(* Logix 5000 project; controller Turck_IOLink_All_Full_AOIs_V0_1 vendor 1 type 14 code 176 rev 32.11; software revision 32.00; part 7 of 7 *)
(* tags used below, declared in another part *)
   Port : INT;
   Write_Application_Specific_Tag : BOOL;
   Universal_IOLink_Info : Universal_IOLink_Info;
   StartupDone : BOOL;
   Done : DINT;
   Error : DINT;
   Active : DINT;
   Pending : DINT;
   Pending_or_Active : DINT;
   MyTicketNum : DINT[32];
   DoneCount : DINT;
   Status : DINT;
   ErrorCount : DINT;
   Prev_Vendor_ID : INT;
   Write_ONS : DINT;
   WriteRequest : DINT;
(* Universal_Device_Info, continued *)

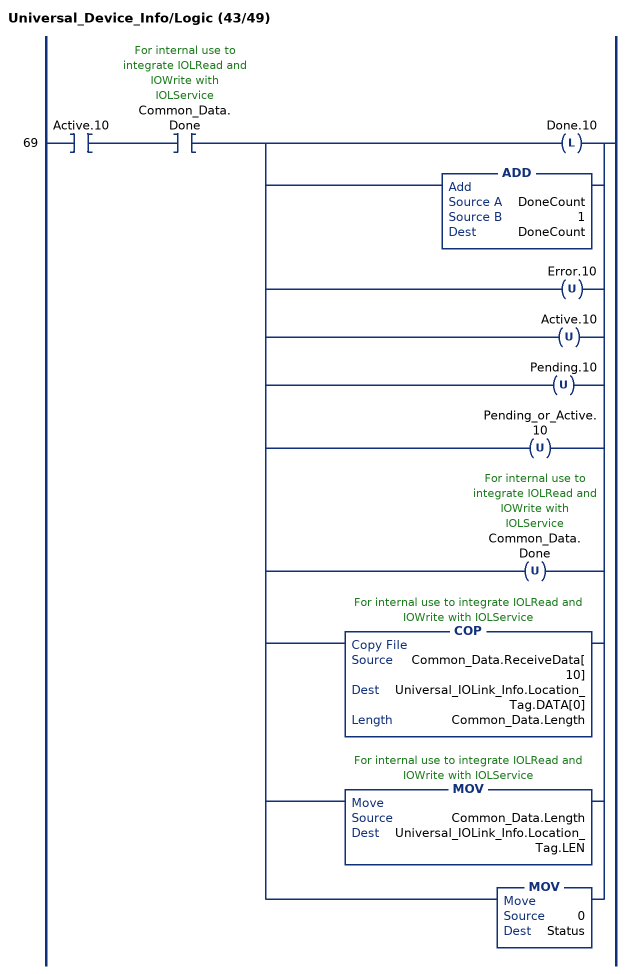
   [picture p146: Universal_Device_Info/Logic rungs 69-69]
   69: XIC(Active.10)XIC(Common_Data.Done)[OTL(Done.10) ,ADD(DoneCount,1,DoneCount) ,OTU(Error.10) ,OTU(Active.10) ,OTU(Pending.10) ,OTU(Pending_or_Active.10) ,OTU(Common_Data.Done) ,COP(Common_Data.ReceiveData[10],Universal_IOLink_Info.Location_Tag.DATA[0],Common_Data.Length) ,MOV(Common_Data.Length,Universal_IOLink_Info.Location_Tag.LEN) ,MOV(0,Status) ];
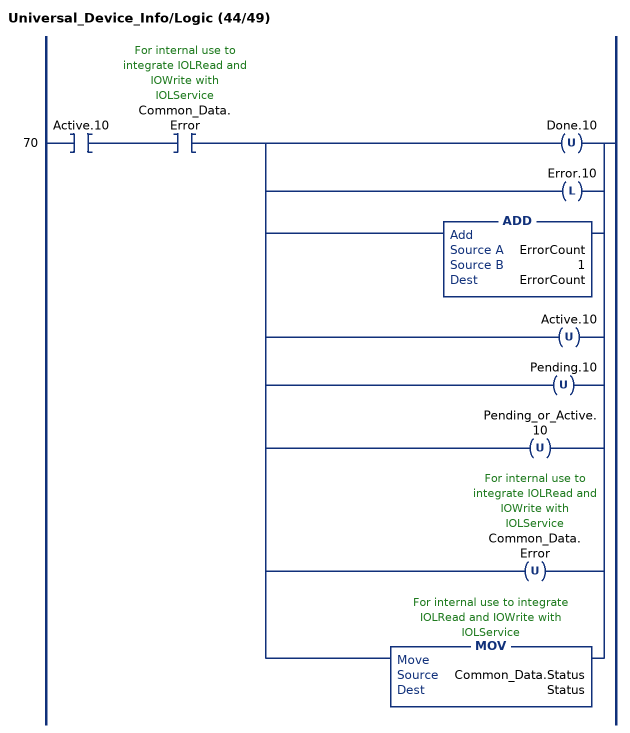
   70: XIC(Active.10)XIC(Common_Data.Error)[OTU(Done.10) ,OTL(Error.10) ,ADD(ErrorCount,1,ErrorCount) ,OTU(Active.10) ,OTU(Pending.10) ,OTU(Pending_or_Active.10) ,OTU(Common_Data.Error) ,MOV(Common_Data.Status,Status) ];
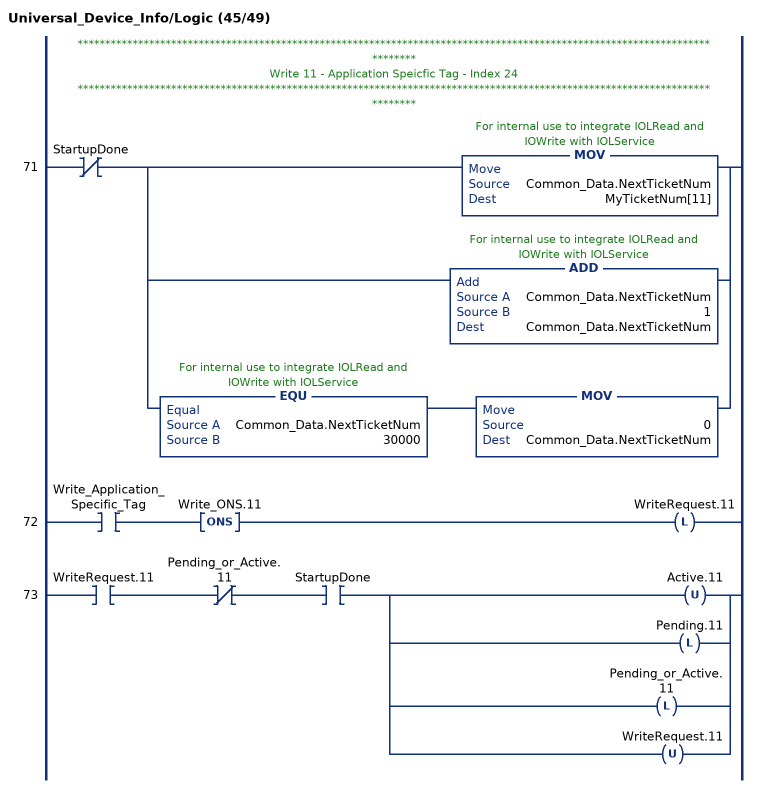
   // ***************************************************************************************************************************
   // Write 11 - Application Speicfic Tag - Index 24
   // ***************************************************************************************************************************
   71: XIO(StartupDone)[MOV(Common_Data.NextTicketNum,MyTicketNum[11]) ,ADD(Common_Data.NextTicketNum,1,Common_Data.NextTicketNum) ,EQU(Common_Data.NextTicketNum,30000) MOV(0,Common_Data.NextTicketNum) ];
   72: XIC(Write_Application_Specific_Tag)ONS(Write_ONS.11)OTL(WriteRequest.11);
   73: XIC(WriteRequest.11)XIO(Pending_or_Active.11)XIC(StartupDone)[OTU(Active.11) ,OTL(Pending.11) ,OTL(Pending_or_Active.11) ,OTU(WriteRequest.11) ];
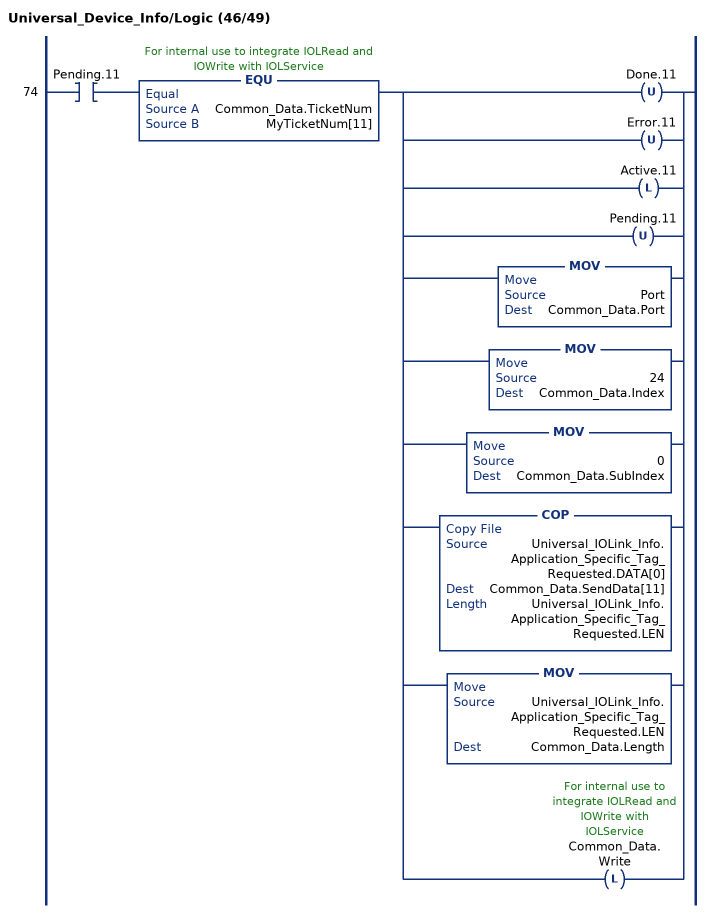
   74: XIC(Pending.11)EQU(Common_Data.TicketNum,MyTicketNum[11])[OTU(Done.11) ,OTU(Error.11) ,OTL(Active.11) ,OTU(Pending.11) ,MOV(Port,Common_Data.Port) ,MOV(24,Common_Data.Index) ,MOV(0,Common_Data.SubIndex) ,COP(Universal_IOLink_Info.Application_Specific_Tag_Requested.DATA[0],Common_Data.SendData[11],Universal_IOLink_Info.Application_Specific_Tag_Requested.LEN) ,MOV(Universal_IOLink_Info.Application_Specific_Tag_Requested.LEN,Common_Data.Length) ,OTL(Common_Data.Write) ];
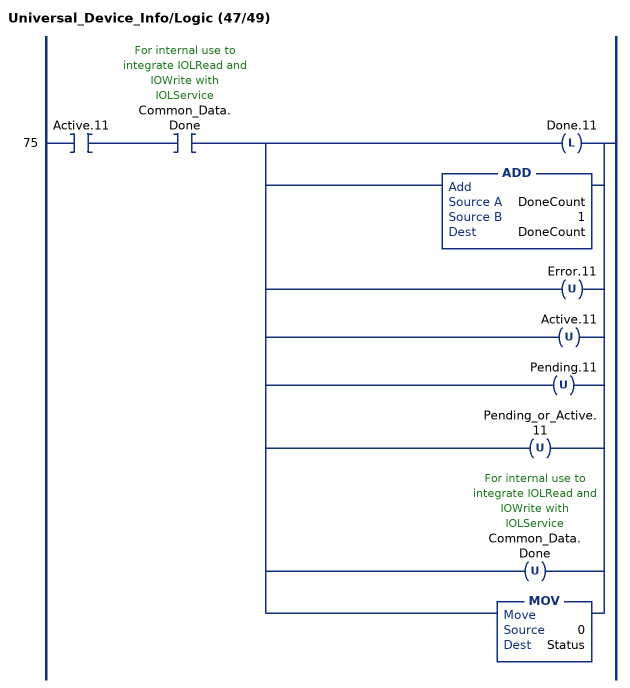
   75: XIC(Active.11)XIC(Common_Data.Done)[OTL(Done.11) ,ADD(DoneCount,1,DoneCount) ,OTU(Error.11) ,OTU(Active.11) ,OTU(Pending.11) ,OTU(Pending_or_Active.11) ,OTU(Common_Data.Done) ,MOV(0,Status) ];
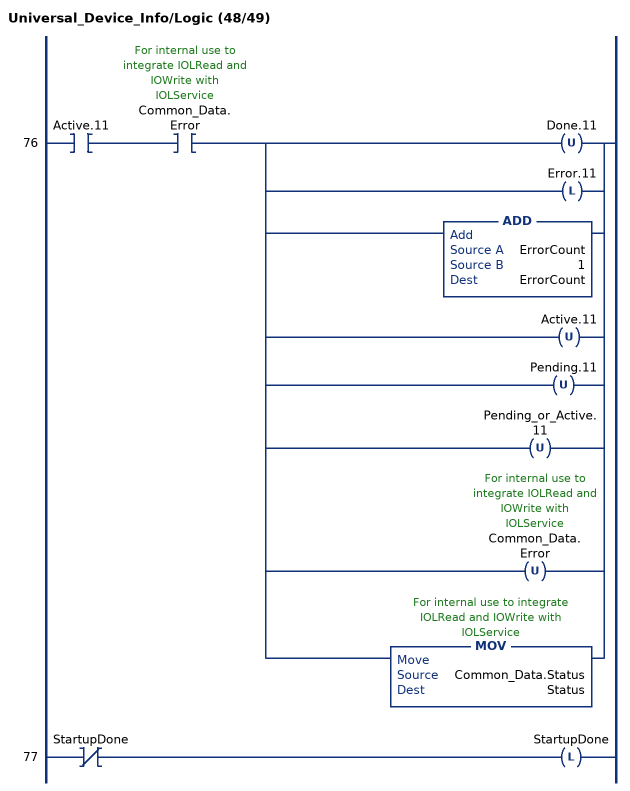
   76: XIC(Active.11)XIC(Common_Data.Error)[OTU(Done.11) ,OTL(Error.11) ,ADD(ErrorCount,1,ErrorCount) ,OTU(Active.11) ,OTU(Pending.11) ,OTU(Pending_or_Active.11) ,OTU(Common_Data.Error) ,MOV(Common_Data.Status,Status) ];
   77: XIO(StartupDone)OTL(StartupDone);
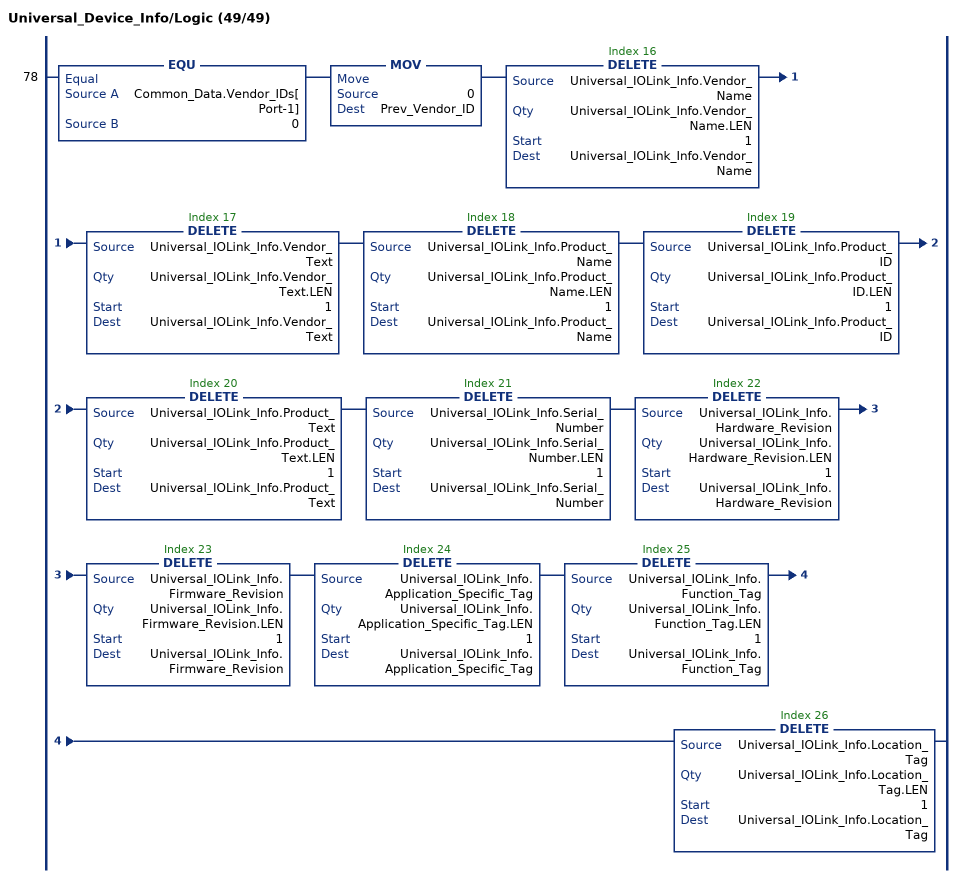
   78: EQU(Common_Data.Vendor_IDs[Port-1],0)MOV(0,Prev_Vendor_ID)DELETE(Universal_IOLink_Info.Vendor_Name,Universal_IOLink_Info.Vendor_Name.LEN,1,Universal_IOLink_Info.Vendor_Name)DELETE(Universal_IOLink_Info.Vendor_Text,Universal_IOLink_Info.Vendor_Text.LEN,1,Universal_IOLink_Info.Vendor_Text)DELETE(Universal_IOLink_Info.Product_Name,Universal_IOLink_Info.Product_Name.LEN,1,Universal_IOLink_Info.Product_Name)DELETE(Universal_IOLink_Info.Product_ID,Universal_IOLink_Info.Product_ID.LEN,1,Universal_IOLink_Info.Product_ID)DELETE(Universal_IOLink_Info.Product_Text,Universal_IOLink_Info.Product_Text.LEN,1,Universal_IOLink_Info.Product_Text)DELETE(Universal_IOLink_Info.Serial_Number,Universal_IOLink_Info.Serial_Number.LEN,1,Universal_IOLink_Info.Serial_Number)DELETE(Universal_IOLink_Info.Hardware_Revision,Universal_IOLink_Info.Hardware_Revision.LEN,1,Universal_IOLink_Info.Hardware_Revision)DELETE(Universal_IOLink_Info.Firmware_Revision,Universal_IOLink_Info.Firmware_Revision.LEN,1,Universal_IOLink_Info.Firmware_Revision)DELETE(Universal_IOLink_Info.Application_Specific_Tag,Universal_IOLink_Info.Application_Specific_Tag.LEN,1,Universal_IOLink_Info.Application_Specific_Tag)DELETE(Universal_IOLink_Info.Function_Tag,Universal_IOLink_Info.Function_Tag.LEN,1,Universal_IOLink_Info.Function_Tag)DELETE(Universal_IOLink_Info.Location_Tag,Universal_IOLink_Info.Location_Tag.LEN,1,Universal_IOLink_Info.Location_Tag);
END_ROUTINE

ROUTINE Prescan   (* ladder *)
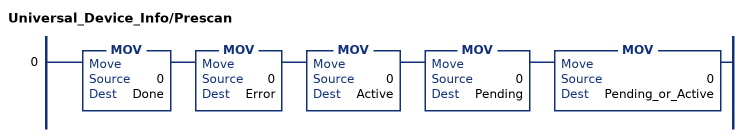
   0: MOV(0,Done)MOV(0,Error)MOV(0,Active)MOV(0,Pending)MOV(0,Pending_or_Active);
END_ROUTINE
END_ADD_ON_INSTRUCTION

VAR_GLOBAL   (* controller tags *)
   Common_Data : Turck_IOLink_Common_Data := (Port := 128, Index := -1, SubIndex := 68, Length := 224, TicketNum := 7, NextTicketNum := 13, SendData[0] := -1, SendData[1] := -1, SendData[2] := 68);
   IOL_READ_MSG : MESSAGE;
        MessageParameters(ServiceCode := 16#004b, LocalElement := Common_Data.SendData, DestinationTag := Common_Data.ReceiveData, ...)
   IOL_WRITE_MSG : MESSAGE;
        MessageParameters(ServiceCode := 16#004c, LocalElement := Common_Data.SendData, DestinationTag := Common_Data.ReceiveData, ...)
   TBEN_100_8IOL_AOI : TBEN_Lx_8IOL_AOI := (DeviceStatus := 16384);
END_VAR

PROGRAM MainProgram   (* main routine MainRoutine *)

ROUTINE MainRoutine   (* ladder *)
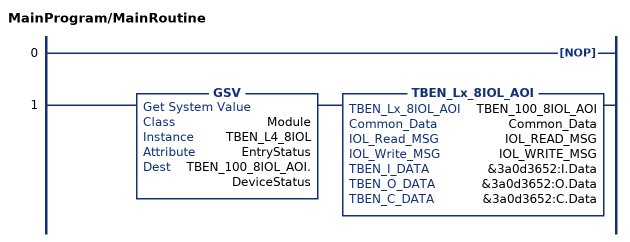
   0: NOP();
   1: GSV(Module,TBEN_L4_8IOL,EntryStatus,TBEN_100_8IOL_AOI.DeviceStatus)TBEN_Lx_8IOL_AOI(TBEN_100_8IOL_AOI,Common_Data,IOL_READ_MSG,IOL_WRITE_MSG,&3a0d3652:I.Data,&3a0d3652:O.Data,&3a0d3652:C.Data);
END_ROUTINE
END_PROGRAM

PROGRAM SafetyProgram   (* main routine MainRoutine, safety *)

ROUTINE MainRoutine   (* ladder *)
END_ROUTINE
END_PROGRAM
